{library PRIVATE}
(*
This is the session handler for all session blocks.
This structure can not be used outside of the CommunicationStructure.
Do not change any values inside the structure instead use existing function blocks to manipulate the data.
*)

TYPE SessionData :
STRUCT
	_Locked:			BOOL:=FALSE;				(* A session lock for this struct *)
	_SessionBussy:		BOOL:=FALSE;				(* If session is bussy sending data *)
	_SessionID:			INT:=0;						(* Session ID that locked this *)
	_SessionCounter:	INT:=0;						(* Sesion counter *)
END_STRUCT
END_TYPE

(* stored: Version 1.1.0.1, ProductVersion 3.1.4024.2
   DUT SessionData: Id {67918ffa-707b-49e5-8422-b837a16a6bdc} *)
